FUNCTION_BLOCK FB_Integer
VAR_INPUT
    nInput  : INT;
END_VAR
VAR_OUTPUT
    nResult : INT;
END_VAR

nResult := nInput + 1;

END_FUNCTION_BLOCK

(* stored: Version 1.1.0.1, ProductVersion 3.1.4024.10
   POU FB_Integer: KindOfPOU Element *)
